(* IEC 61131-3 sources: Std_PalletMover/Class/HmiOption1_MqttCommuncation, 1 file *)

(* ---- HmiOption1_MqttCommuncation.st ---- *)
(*!
<Class
	Name               = "HmiOption1_MqttCommuncation"
	Revision           = "0.0"
	RealtimeTask       = "false"
	CyclicTask         = "false"
	BackgroundTask     = "false"
	Sigmatek           = "false"
	OSInterface        = "false"
	HighPriority       = "false"
	Automatic          = "false"
	UpdateMode         = "Prescan"
	SharedCommandTable = "true"
	Objectsize         = "(1020,120)">
	<Channels>
		<Server Name="ClassSvr" Visualized="false" Initialize="false" WriteProtected="true" Retentive="false"/>
		<Server Name="HmiInterface" Class="I_Hmi" Visualized="false" Initialize="false" WriteProtected="true" Retentive="false"/>
	</Channels>
	<Network Name="HmiOption1_MqttCommuncation">
		<!-- List of Components in this network -->
		<Components>
		</Components>
		<Comments>
		</Comments>
		<!-- List of Connections in this network -->
		<Connections>
		</Connections>
		<!-- Headerfiles -->
		<Options>
		</Options>
	</Network>
</Class>
*)
HmiOption1_MqttCommuncation : CLASS
  //Servers:
	ClassSvr 	: SvrChCmd_DINT;
	HmiInterface 	: SvrChCmd_DINT;
  //Clients:
  //Variables:
  //Functions:

	FUNCTION VIRTUAL GLOBAL HmiInterface::Read
		VAR_OUTPUT
			output (EAX) 	: DINT;
		END_VAR;
  //Tables:
	FUNCTION @STD
		VAR_OUTPUT
			ret_code	: CONFSTATES;
		END_VAR;
	FUNCTION GLOBAL TAB @CT_;
END_CLASS;

FUNCTION VIRTUAL GLOBAL HmiOption1_MqttCommuncation::HmiInterface::Read
	VAR_OUTPUT
		output (EAX) 	: DINT;
	END_VAR

	HmiInterface := I_Hmi1.ClassSvr.Read();
	output := HmiInterface;

END_FUNCTION
